{attribute addProperty BoxType "AT2050-0500-0017"}
{attribute addProperty Id "A_0096_AT2025_5250_0017_AT2025_5250AT2025_C5E5984862678.25"}
{attribute addProperty CRC "2830470941"}
{attribute addProperty SizeInBites "626"}
{attribute addProperty SizeInBytes "78.25"}
TYPE A_0048_AT2050_0500_0017_A8B58F1D EXTENDS AT2050_BA5A9548 :
STRUCT
	{attribute addProperty Name "A_0096_AT2025_5250_0017_AT2025_5250"}
	A_0096_AT2025_5250_0017_AT2025_5250 : AT2025_C5E59848;
END_STRUCT
END_TYPE

(* stored: Version 1.2.0.0, ProductVersion 3.1.4024.9
   DUT A_0048_AT2050_0500_0017_A8B58F1D: Id {df0b04dc-dc46-4c3d-a59b-1eacac2759ac} *)
